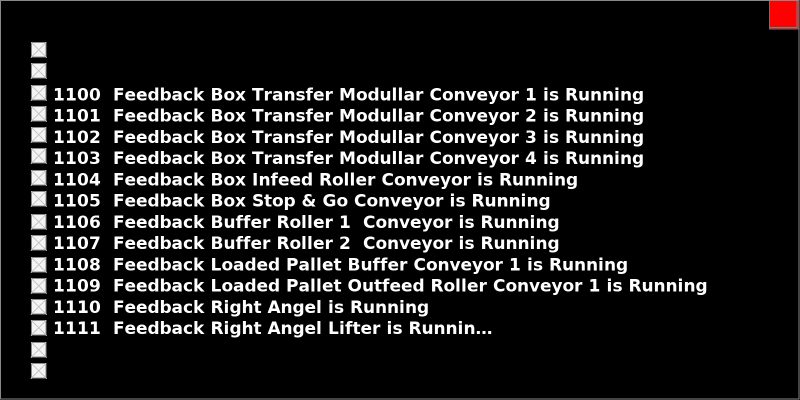
VISUALIZATION P2_DI2  // 800x400, background image 
    ImageSwitcher (31,42 15x15), variable: InputOutput_GVL.Digital_Input[17], behaviour: TOGGLE
    Label (50,16 720x391), "1100 Feedback Box Transfer Modullar Conveyor 1 is Running 1101 Feedback Box Transfer Modullar Conveyor 2 is Running 1102 Feedback Box Transfer Modullar Conveyor 3 is Running 1103 Feedback Box Transfer Modullar Conveyor 4 is Running 1104 Feedback Box Infeed Roller Conveyor is Running 1105 Feedback Box Stop & Go Conveyor is Running 1106 Feedback Buffer Roller 1 Conveyor is Running 1107 Feedback Buffer Roller 2 Conveyor is Running 1108 Feedback Loaded Pallet Buffer Conveyor 1 is Running 1109 Feedback Loaded Pallet Outfeed Roller Conveyor 1 is Running 1110 Feedback Right Angel is Running 1111 Feedback Right Angel Lifter is Running 1112 Feedback Loaded Pallet Outfeed Roller Conveyor 2 is Running 1113 Feedback Loaded Pallet Outfeed Roller Conveyor 3 is Running 1114 Feedback Loaded Pallet Outfeed Roller Conveyor 4 is Running 1115 Feedback Loaded Pallet Buffer 2 is Running"
    ImageSwitcher (31,63 15x15), variable: InputOutput_GVL.Digital_Input[18], behaviour: TOGGLE
    ImageSwitcher (31,85 15x15), variable: InputOutput_GVL.Digital_Input[19], behaviour: TOGGLE
    ImageSwitcher (31,106 15x15), variable: InputOutput_GVL.Digital_Input[20], behaviour: TOGGLE
    ImageSwitcher (31,127 15x15), variable: InputOutput_GVL.Digital_Input[21], behaviour: TOGGLE
    ImageSwitcher (31,148 15x15), variable: InputOutput_GVL.Digital_Input[22], behaviour: TOGGLE
    ImageSwitcher (31,170 15x15), variable: InputOutput_GVL.Digital_Input[23], behaviour: TOGGLE
    ImageSwitcher (31,191 15x15), variable: InputOutput_GVL.Digital_Input[24], behaviour: TOGGLE
    ImageSwitcher (31,214 15x15), variable: InputOutput_GVL.Digital_Input[25], behaviour: TOGGLE
    ImageSwitcher (31,235 15x15), variable: InputOutput_GVL.Digital_Input[26], behaviour: TOGGLE
    ImageSwitcher (31,257 15x15), variable: InputOutput_GVL.Digital_Input[27], behaviour: TOGGLE
    ImageSwitcher (31,278 15x15), variable: InputOutput_GVL.Digital_Input[28], behaviour: TOGGLE
    ImageSwitcher (31,299 15x15), variable: InputOutput_GVL.Digital_Input[29], behaviour: TOGGLE
    ImageSwitcher (31,320 15x15), variable: InputOutput_GVL.Digital_Input[30], behaviour: TOGGLE
    ImageSwitcher (31,342 15x15), variable: InputOutput_GVL.Digital_Input[31], behaviour: TOGGLE
    ImageSwitcher (31,363 15x15), variable: InputOutput_GVL.Digital_Input[32], behaviour: TOGGLE
    Button (769,-1 30x30), image: VisuSymbols.Symbols.Wrong
        OnMouseClick: CloseDialog Dialog=P2_DI2, Result=OK, NumpadKeypadSet=True
END_VISUALIZATION

(* stored: Version 1.1.0.1, ProductVersion 3.1.4024.12
   Visu P2_DI2: Id {2212f306-b437-4ce9-ba19-2b1e0a223ba6} *)
